(* Logix 5000 project; controller cal1632 1756-L62 rev 16.20; software revision 16.05; part 12 of 57 *)
(* tags used below, declared in another part *)
   AFI : BOOL;
   FAULT : BOOL;
   p01_param_open_oven_temp : REAL;
   p01_param_oven_timer_presets : DINT[32];
   p01_param_process_air_hl : REAL;
   p01_recipe_active : recipe;
   p01_sys_enc : SYS_ENC;
   p01_sys_lc : Limit_Clamp;
   p01r09_open_oven : BOOL;
   p01r09_pb_global_reset : BOOL;
   p01r13_permissive_oxidizer : BOOL;
   p02_dint_from_hmi : hmi_dint;
   p02_real_from_hmi : hmi_real;
   p11_ai_lfl : REAL;
   p11_ai_tc01 : REAL;
   p11_ai_tc02 : REAL;
   p11_ao_cv : REAL;
   p11_di_burner_auto : BOOL;
   p11_di_burner_safeties_ok : BOOL;
   p11_di_exh_flow_ok : BOOL;
   p11_di_flame_failure : BOOL;
   p11_di_flame_on : BOOL;
   p11_di_high_limit_temp_ok : BOOL;
   p11_di_recirc_flow_ok : BOOL;
   p11_di_sp1 : BOOL;
   p11_di_tc01_bo : BOOL;
   p11_di_tc02_bo : BOOL;
   p11_do_enable_burner : BOOL;
   p11_do_rst_flame : BOOL;
   p11_param_fast_to_soak : REAL;
   p11_param_lfl_hhl : REAL;
   p11_param_lfl_hl : REAL;
   p11_param_pid1_ff : REAL;
   p11_param_pid1_kd : REAL;
   p11_param_pid1_ki : REAL;
   p11_param_pid1_kp : REAL;
   p11_param_pid2_ff : REAL;
   p11_param_pid2_kd : REAL;
   p11_param_pid2_ki : REAL;
   p11_param_pid2_kp : REAL;
   p11_param_shutdown_temp : REAL;
   p11_param_soak_to_fast : REAL;
   p11_param_tc01_dev : REAL;
   p11_param_tc01_hl : REAL;
   p11_param_tc01z : REAL;
   p11_param_tc02z : REAL;
   p11_param_zone_pressure : REAL;
   p11r02_shutdown_temp : BOOL;
   p11r02_timer_safe_temp : TIMER[2];
   p11r02_timer_warning : TIMER[4];
   p11r10 : routine;
   p11r10_timer_fault : TIMER[4];
   p11r10_timer_warning : TIMER[4];
   p11r12_Oven_auto_run_on : BOOL;
   p11r16_pid_temp_cv : DINT;
   p11r16_temp_ok : BOOL;
   p11r20 : routine;
   p11r20_safeties_ok : BOOL;
   p11r20_state : DINT;
   p11r20_status : DINT;
   p11r20_timer_fault : TIMER[4];
   p11r20_timer_state_11 : TIMER;
   p11r20_timer_state_3 : TIMER;
   p11r20_timer_state_4 : TIMER;
   p11r20_timer_state_7 : TIMER;
   p11r20_timer_warning : TIMER[4];
   p11r30 : routine;
   p11r30_cv_man_sp : REAL;
   p11r30_pb_auto : BOOL;
   p11r30_pb_manual : BOOL;
   p11r30_pb_zone_off : BOOL;
   p11r30_pb_zone_on : BOOL;
   p11r30_permissive_run : BOOL;
   p11r30_pid_temp : PID;
   p11r30_pid_temp_pv : REAL;
   p11r30_pid_temp_sp : REAL;
   p11r30_pid_temp_sp_error : REAL;
   p11r30_pid_temp_sp_last : REAL;
   p11r30_request_deviation_warning : BOOL;
   p11r30_request_heat : BOOL;
   p11r30_request_heat_last : BOOL;
   p11r30_request_manual : BOOL;
   p11r30_request_PID_shot : BOOL;
   p11r30_request_soak_control : BOOL;
   p11r30_temp_deviation_setpoint : DINT;
   p11r30_timer_fault : TIMER[16];
   p11r30_timer_warning : TIMER[12];
   p11r30_vfds_ok : BOOL;
   p11r31 : routine;
   p11r31_timer_fault : TIMER[5];
   p11r31_timer_warning : TIMER[5];
   p11r32 : routine;
   p11r32_timer_fault : TIMER[5];
   p11r32_timer_warning : TIMER[5];
   p12r30 : routine;
   p23_di_impreg_exhaust_running : BOOL;
   p23_di_impreg_tank_up : BOOL;
   p23r02 : routine;
   p23r13 : routine;
(* P11_Zone_1, continued *)

ROUTINE R10_Parameters   (* ladder *)
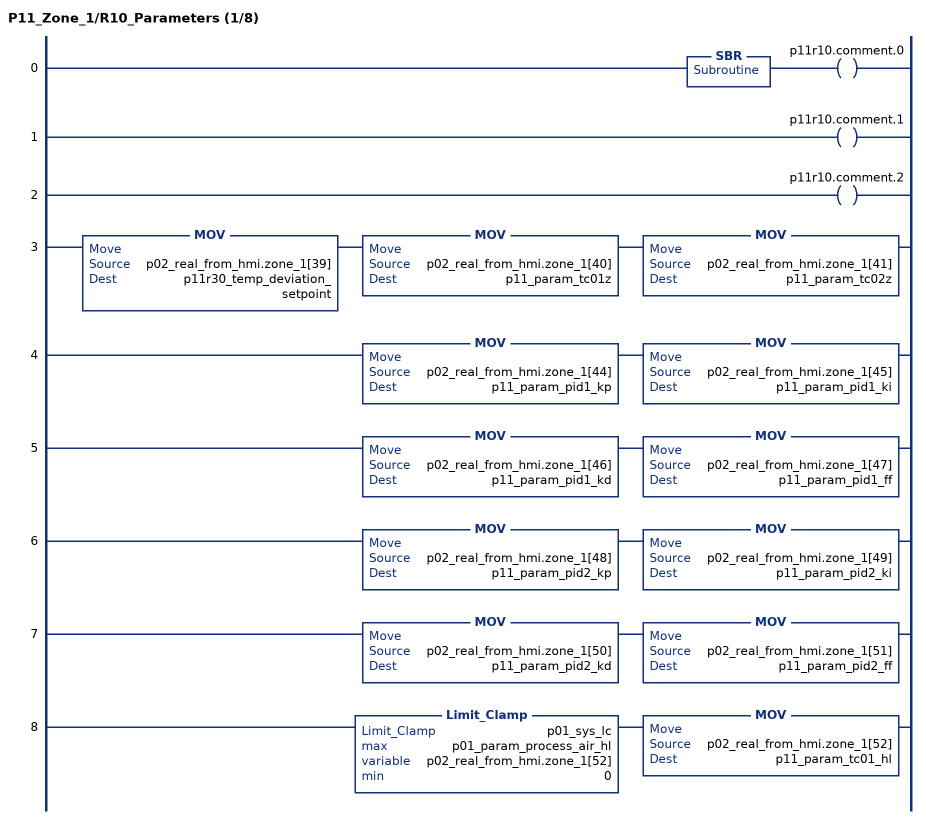
   0: SBR()OTE(p11r10.comment.0);
   1: OTE(p11r10.comment.1);
   2: OTE(p11r10.comment.2);
   3: MOV(p02_real_from_hmi.zone_1[39],p11r30_temp_deviation_setpoint)MOV(p02_real_from_hmi.zone_1[40],p11_param_tc01z)MOV(p02_real_from_hmi.zone_1[41],p11_param_tc02z);
   4: MOV(p02_real_from_hmi.zone_1[44],p11_param_pid1_kp)MOV(p02_real_from_hmi.zone_1[45],p11_param_pid1_ki);
   5: MOV(p02_real_from_hmi.zone_1[46],p11_param_pid1_kd)MOV(p02_real_from_hmi.zone_1[47],p11_param_pid1_ff);
   6: MOV(p02_real_from_hmi.zone_1[48],p11_param_pid2_kp)MOV(p02_real_from_hmi.zone_1[49],p11_param_pid2_ki);
   7: MOV(p02_real_from_hmi.zone_1[50],p11_param_pid2_kd)MOV(p02_real_from_hmi.zone_1[51],p11_param_pid2_ff);
   8: Limit_Clamp(p01_sys_lc,p01_param_process_air_hl,p02_real_from_hmi.zone_1[52],0)MOV(p02_real_from_hmi.zone_1[52],p11_param_tc01_hl);
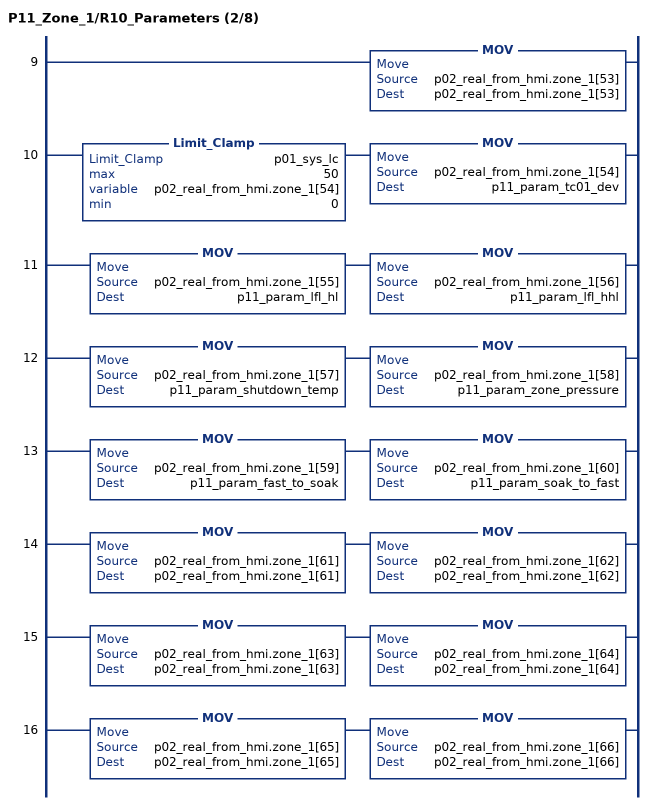
   9: MOV(p02_real_from_hmi.zone_1[53],p02_real_from_hmi.zone_1[53]);
   10: Limit_Clamp(p01_sys_lc,50,p02_real_from_hmi.zone_1[54],0)MOV(p02_real_from_hmi.zone_1[54],p11_param_tc01_dev);
   11: MOV(p02_real_from_hmi.zone_1[55],p11_param_lfl_hl)MOV(p02_real_from_hmi.zone_1[56],p11_param_lfl_hhl);
   12: MOV(p02_real_from_hmi.zone_1[57],p11_param_shutdown_temp)MOV(p02_real_from_hmi.zone_1[58],p11_param_zone_pressure);
   13: MOV(p02_real_from_hmi.zone_1[59],p11_param_fast_to_soak)MOV(p02_real_from_hmi.zone_1[60],p11_param_soak_to_fast);
   14: MOV(p02_real_from_hmi.zone_1[61],p02_real_from_hmi.zone_1[61])MOV(p02_real_from_hmi.zone_1[62],p02_real_from_hmi.zone_1[62]);
   15: MOV(p02_real_from_hmi.zone_1[63],p02_real_from_hmi.zone_1[63])MOV(p02_real_from_hmi.zone_1[64],p02_real_from_hmi.zone_1[64]);
   16: MOV(p02_real_from_hmi.zone_1[65],p02_real_from_hmi.zone_1[65])MOV(p02_real_from_hmi.zone_1[66],p02_real_from_hmi.zone_1[66]);
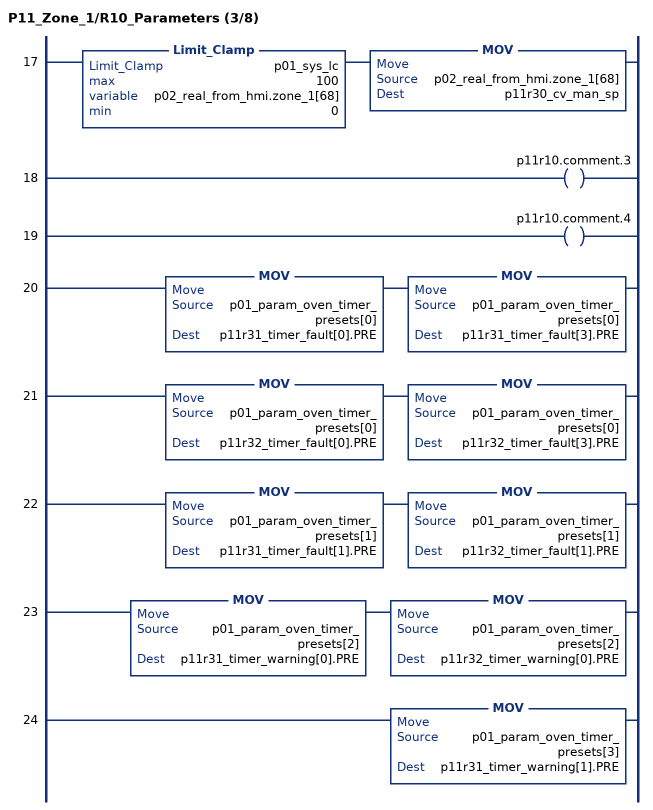
   17: Limit_Clamp(p01_sys_lc,100,p02_real_from_hmi.zone_1[68],0)MOV(p02_real_from_hmi.zone_1[68],p11r30_cv_man_sp);
   18: OTE(p11r10.comment.3);
   19: OTE(p11r10.comment.4);
   20: MOV(p01_param_oven_timer_presets[0],p11r31_timer_fault[0].PRE)MOV(p01_param_oven_timer_presets[0],p11r31_timer_fault[3].PRE);
   21: MOV(p01_param_oven_timer_presets[0],p11r32_timer_fault[0].PRE)MOV(p01_param_oven_timer_presets[0],p11r32_timer_fault[3].PRE);
   22: MOV(p01_param_oven_timer_presets[1],p11r31_timer_fault[1].PRE)MOV(p01_param_oven_timer_presets[1],p11r32_timer_fault[1].PRE);
   23: MOV(p01_param_oven_timer_presets[2],p11r31_timer_warning[0].PRE)MOV(p01_param_oven_timer_presets[2],p11r32_timer_warning[0].PRE);
   24: MOV(p01_param_oven_timer_presets[3],p11r31_timer_warning[1].PRE);
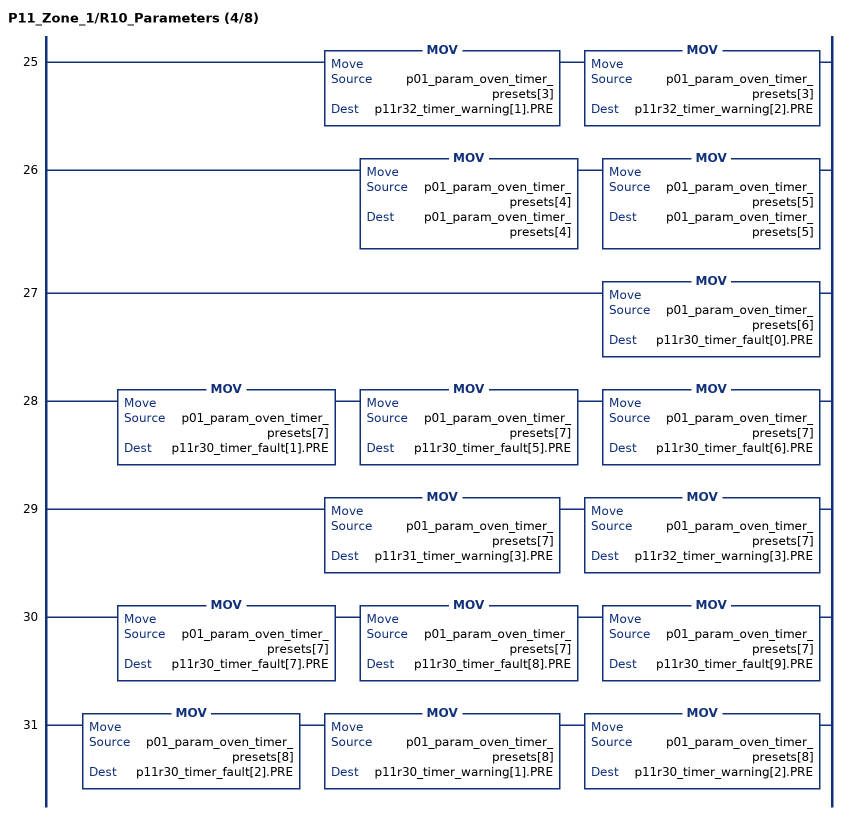
   25: MOV(p01_param_oven_timer_presets[3],p11r32_timer_warning[1].PRE)MOV(p01_param_oven_timer_presets[3],p11r32_timer_warning[2].PRE);
   26: MOV(p01_param_oven_timer_presets[4],p01_param_oven_timer_presets[4])MOV(p01_param_oven_timer_presets[5],p01_param_oven_timer_presets[5]);
   27: MOV(p01_param_oven_timer_presets[6],p11r30_timer_fault[0].PRE);
   28: MOV(p01_param_oven_timer_presets[7],p11r30_timer_fault[1].PRE)MOV(p01_param_oven_timer_presets[7],p11r30_timer_fault[5].PRE)MOV(p01_param_oven_timer_presets[7],p11r30_timer_fault[6].PRE);
   29: MOV(p01_param_oven_timer_presets[7],p11r31_timer_warning[3].PRE)MOV(p01_param_oven_timer_presets[7],p11r32_timer_warning[3].PRE);
   30: MOV(p01_param_oven_timer_presets[7],p11r30_timer_fault[7].PRE)MOV(p01_param_oven_timer_presets[7],p11r30_timer_fault[8].PRE)MOV(p01_param_oven_timer_presets[7],p11r30_timer_fault[9].PRE);
   31: MOV(p01_param_oven_timer_presets[8],p11r30_timer_fault[2].PRE)MOV(p01_param_oven_timer_presets[8],p11r30_timer_warning[1].PRE)MOV(p01_param_oven_timer_presets[8],p11r30_timer_warning[2].PRE);
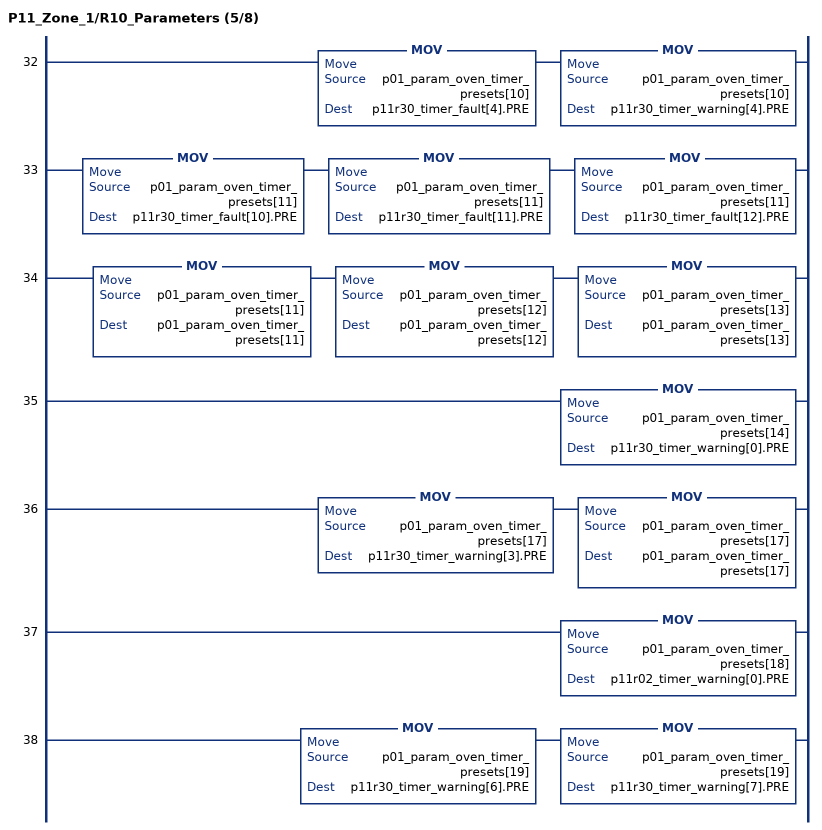
   32: MOV(p01_param_oven_timer_presets[10],p11r30_timer_fault[4].PRE)MOV(p01_param_oven_timer_presets[10],p11r30_timer_warning[4].PRE);
   33: MOV(p01_param_oven_timer_presets[11],p11r30_timer_fault[10].PRE)MOV(p01_param_oven_timer_presets[11],p11r30_timer_fault[11].PRE)MOV(p01_param_oven_timer_presets[11],p11r30_timer_fault[12].PRE);
   34: MOV(p01_param_oven_timer_presets[11],p01_param_oven_timer_presets[11])MOV(p01_param_oven_timer_presets[12],p01_param_oven_timer_presets[12])MOV(p01_param_oven_timer_presets[13],p01_param_oven_timer_presets[13]);
   35: MOV(p01_param_oven_timer_presets[14],p11r30_timer_warning[0].PRE);
   36: MOV(p01_param_oven_timer_presets[17],p11r30_timer_warning[3].PRE)MOV(p01_param_oven_timer_presets[17],p01_param_oven_timer_presets[17]);
   37: MOV(p01_param_oven_timer_presets[18],p11r02_timer_warning[0].PRE);
   38: MOV(p01_param_oven_timer_presets[19],p11r30_timer_warning[6].PRE)MOV(p01_param_oven_timer_presets[19],p11r30_timer_warning[7].PRE);
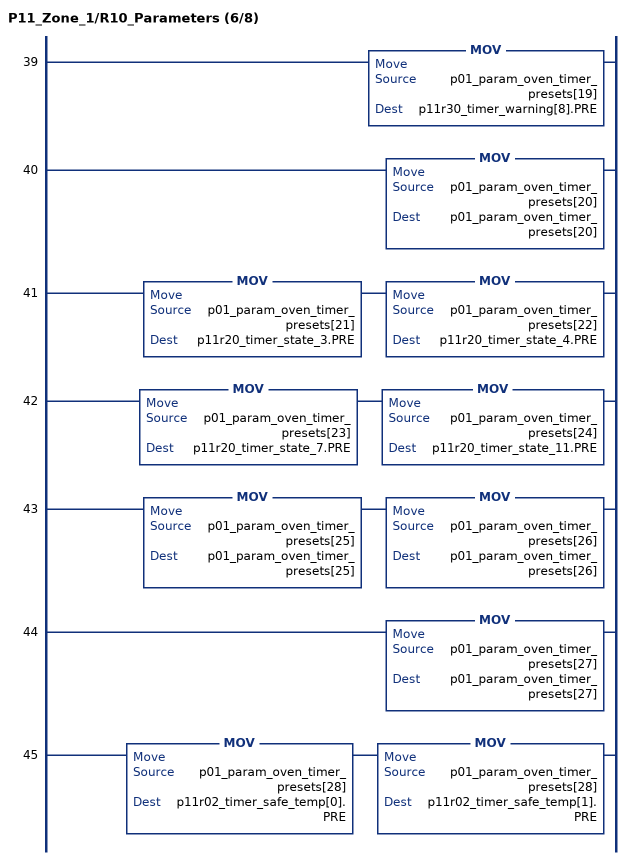
   39: MOV(p01_param_oven_timer_presets[19],p11r30_timer_warning[8].PRE);
   40: MOV(p01_param_oven_timer_presets[20],p01_param_oven_timer_presets[20]);
   41: MOV(p01_param_oven_timer_presets[21],p11r20_timer_state_3.PRE)MOV(p01_param_oven_timer_presets[22],p11r20_timer_state_4.PRE);
   42: MOV(p01_param_oven_timer_presets[23],p11r20_timer_state_7.PRE)MOV(p01_param_oven_timer_presets[24],p11r20_timer_state_11.PRE);
   43: MOV(p01_param_oven_timer_presets[25],p01_param_oven_timer_presets[25])MOV(p01_param_oven_timer_presets[26],p01_param_oven_timer_presets[26]);
   44: MOV(p01_param_oven_timer_presets[27],p01_param_oven_timer_presets[27]);
   45: MOV(p01_param_oven_timer_presets[28],p11r02_timer_safe_temp[0].PRE)MOV(p01_param_oven_timer_presets[28],p11r02_timer_safe_temp[1].PRE);
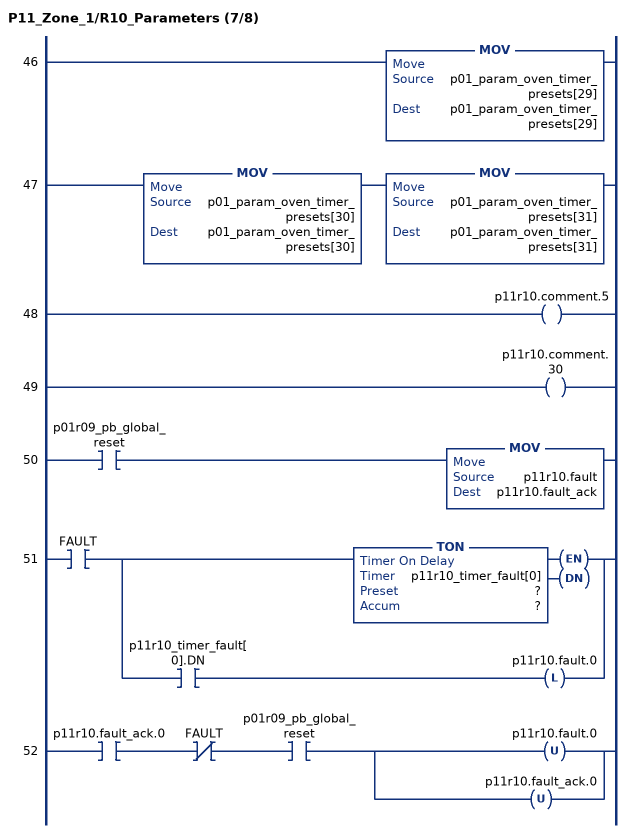
   46: MOV(p01_param_oven_timer_presets[29],p01_param_oven_timer_presets[29]);
   47: MOV(p01_param_oven_timer_presets[30],p01_param_oven_timer_presets[30])MOV(p01_param_oven_timer_presets[31],p01_param_oven_timer_presets[31]);
   48: OTE(p11r10.comment.5);
   49: OTE(p11r10.comment.30);
   50: XIC(p01r09_pb_global_reset)MOV(p11r10.fault,p11r10.fault_ack);
   51: XIC(FAULT)[TON(p11r10_timer_fault[0],?,?) ,XIC(p11r10_timer_fault[0].DN) OTL(p11r10.fault.0) ];
   52: XIC(p11r10.fault_ack.0)XIO(FAULT)XIC(p01r09_pb_global_reset)[OTU(p11r10.fault.0) ,OTU(p11r10.fault_ack.0) ];
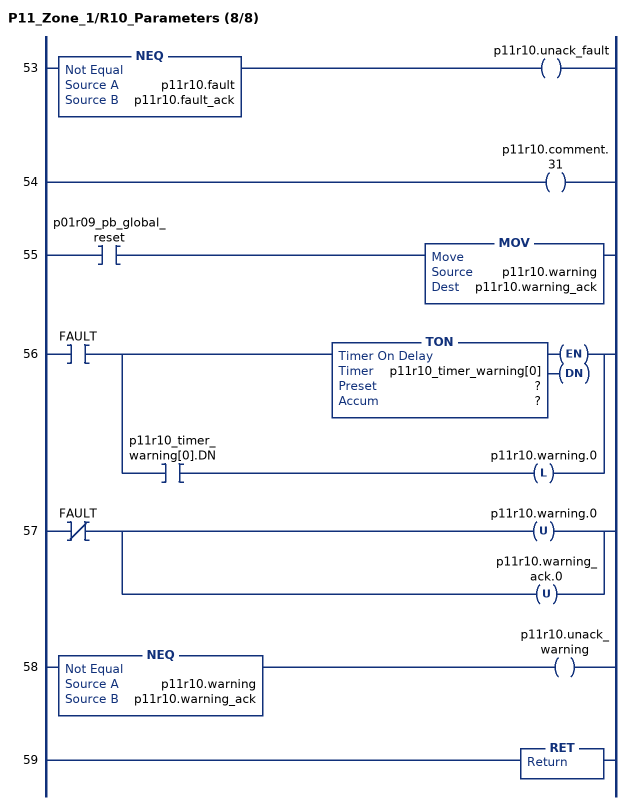
   53: NEQ(p11r10.fault,p11r10.fault_ack)OTE(p11r10.unack_fault);
   54: OTE(p11r10.comment.31);
   55: XIC(p01r09_pb_global_reset)MOV(p11r10.warning,p11r10.warning_ack);
   56: XIC(FAULT)[TON(p11r10_timer_warning[0],?,?) ,XIC(p11r10_timer_warning[0].DN) OTL(p11r10.warning.0) ];
   57: XIO(FAULT)[OTU(p11r10.warning.0) ,OTU(p11r10.warning_ack.0) ];
   58: NEQ(p11r10.warning,p11r10.warning_ack)OTE(p11r10.unack_warning);
   59: RET();
END_ROUTINE

ROUTINE R20_Temp_Sequence   (* ladder *)
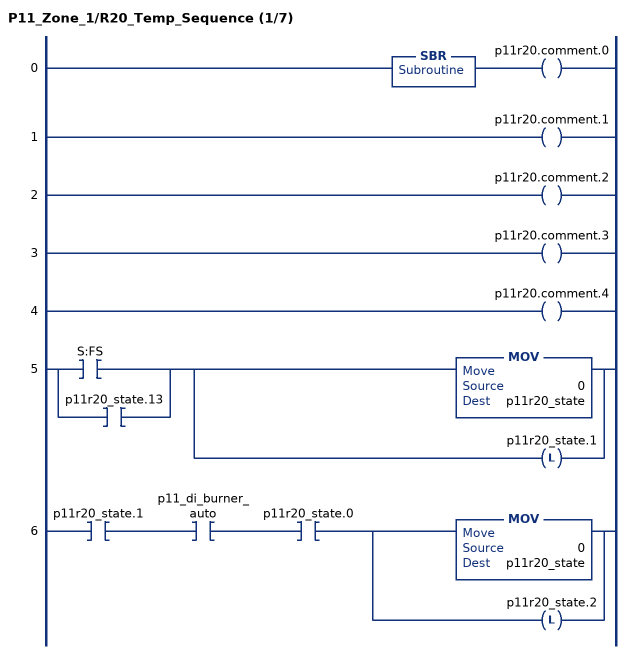
   0: SBR()OTE(p11r20.comment.0);
   1: OTE(p11r20.comment.1);
   2: OTE(p11r20.comment.2);
   3: OTE(p11r20.comment.3);
   4: OTE(p11r20.comment.4);
   5: [XIC(S:FS) ,XIC(p11r20_state.13) ][MOV(0,p11r20_state) ,OTL(p11r20_state.1) ];
   6: XIC(p11r20_state.1)XIC(p11_di_burner_auto)XIC(p11r20_state.0)[MOV(0,p11r20_state) ,OTL(p11r20_state.2) ];
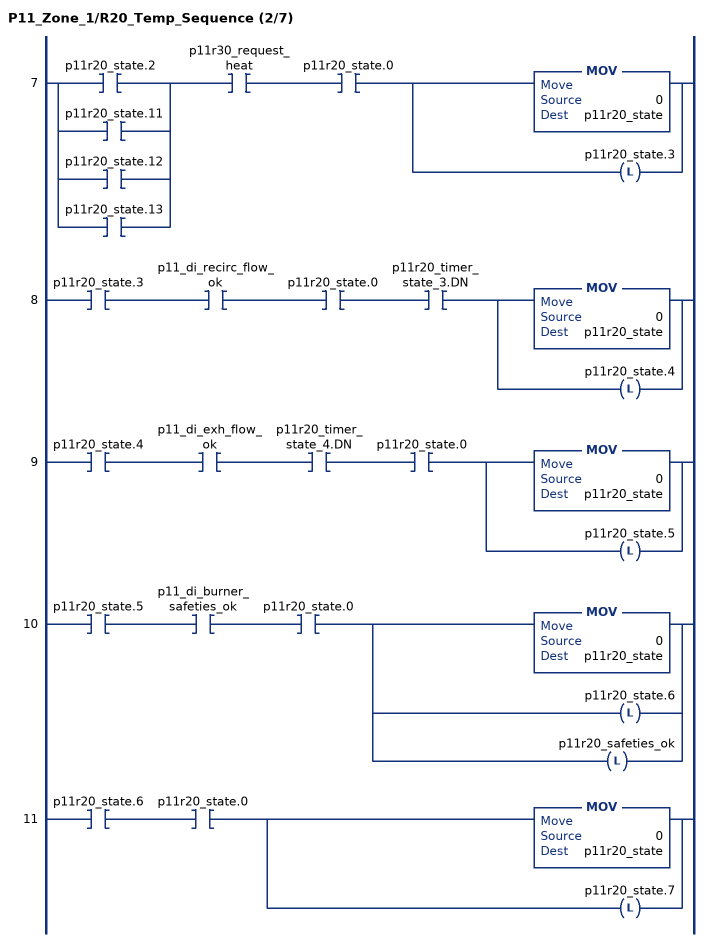
   7: [XIC(p11r20_state.2) ,XIC(p11r20_state.11) ,XIC(p11r20_state.12) ,XIC(p11r20_state.13) ]XIC(p11r30_request_heat)XIC(p11r20_state.0)[MOV(0,p11r20_state) ,OTL(p11r20_state.3) ];
   8: XIC(p11r20_state.3)XIC(p11_di_recirc_flow_ok)XIC(p11r20_state.0)XIC(p11r20_timer_state_3.DN)[MOV(0,p11r20_state) ,OTL(p11r20_state.4) ];
   9: XIC(p11r20_state.4)XIC(p11_di_exh_flow_ok)XIC(p11r20_timer_state_4.DN)XIC(p11r20_state.0)[MOV(0,p11r20_state) ,OTL(p11r20_state.5) ];
   10: XIC(p11r20_state.5)XIC(p11_di_burner_safeties_ok)XIC(p11r20_state.0)[MOV(0,p11r20_state) ,OTL(p11r20_state.6) ,OTL(p11r20_safeties_ok) ];
   11: XIC(p11r20_state.6)XIC(p11r20_state.0)[MOV(0,p11r20_state) ,OTL(p11r20_state.7) ];
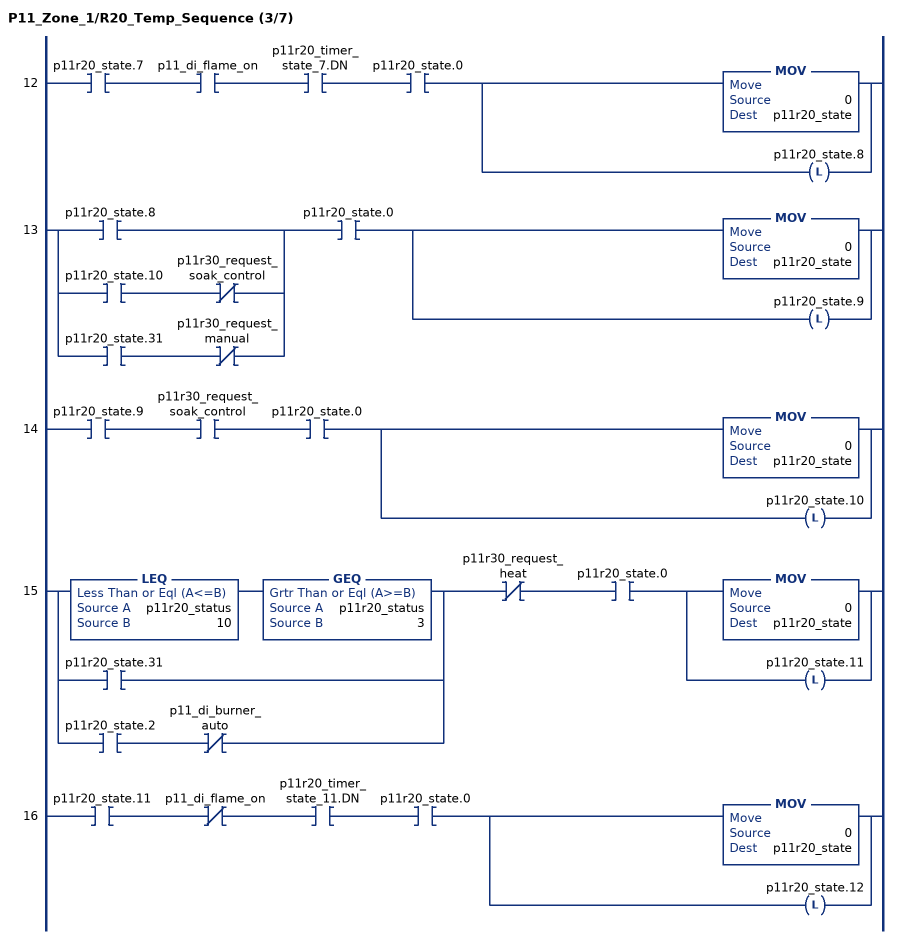
   12: XIC(p11r20_state.7)XIC(p11_di_flame_on)XIC(p11r20_timer_state_7.DN)XIC(p11r20_state.0)[MOV(0,p11r20_state) ,OTL(p11r20_state.8) ];
   13: [XIC(p11r20_state.8) ,XIC(p11r20_state.10) XIO(p11r30_request_soak_control) ,XIC(p11r20_state.31) XIO(p11r30_request_manual) ]XIC(p11r20_state.0)[MOV(0,p11r20_state) ,OTL(p11r20_state.9) ];
   14: XIC(p11r20_state.9)XIC(p11r30_request_soak_control)XIC(p11r20_state.0)[MOV(0,p11r20_state) ,OTL(p11r20_state.10) ];
   15: [[LEQ(p11r20_status,10) GEQ(p11r20_status,3) ,XIC(p11r20_state.31) ] ,XIC(p11r20_state.2) XIO(p11_di_burner_auto) ]XIO(p11r30_request_heat)XIC(p11r20_state.0)[MOV(0,p11r20_state) ,OTL(p11r20_state.11) ];
   16: XIC(p11r20_state.11)XIO(p11_di_flame_on)XIC(p11r20_timer_state_11.DN)XIC(p11r20_state.0)[MOV(0,p11r20_state) ,OTL(p11r20_state.12) ];
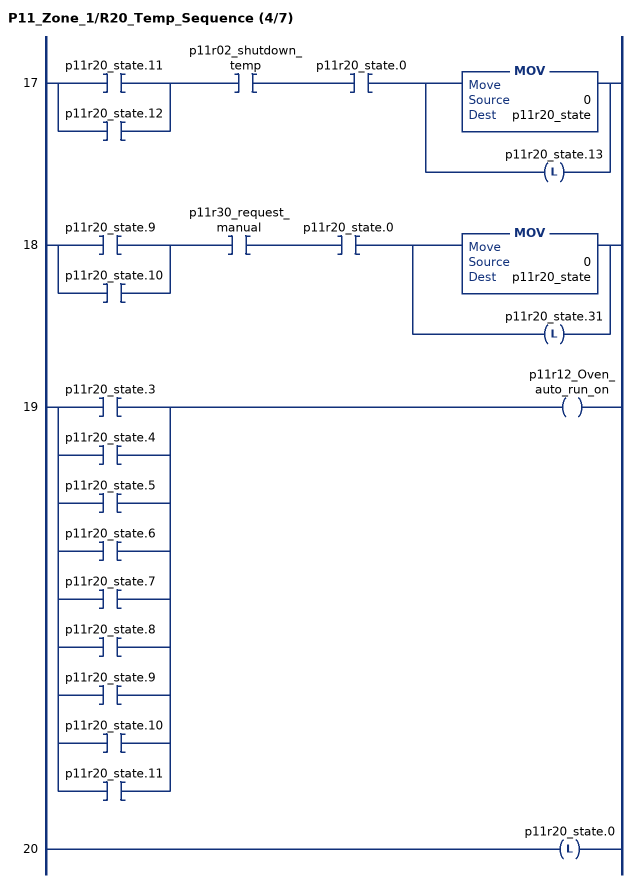
   17: [XIC(p11r20_state.11) ,XIC(p11r20_state.12) ]XIC(p11r02_shutdown_temp)XIC(p11r20_state.0)[MOV(0,p11r20_state) ,OTL(p11r20_state.13) ];
   18: [XIC(p11r20_state.9) ,XIC(p11r20_state.10) ]XIC(p11r30_request_manual)XIC(p11r20_state.0)[MOV(0,p11r20_state) ,OTL(p11r20_state.31) ];
   19: [XIC(p11r20_state.3) ,XIC(p11r20_state.4) ,XIC(p11r20_state.5) ,XIC(p11r20_state.6) ,XIC(p11r20_state.7) ,XIC(p11r20_state.8) ,XIC(p11r20_state.9) ,XIC(p11r20_state.10) ,XIC(p11r20_state.11) ]OTE(p11r12_Oven_auto_run_on);
   20: OTL(p11r20_state.0);
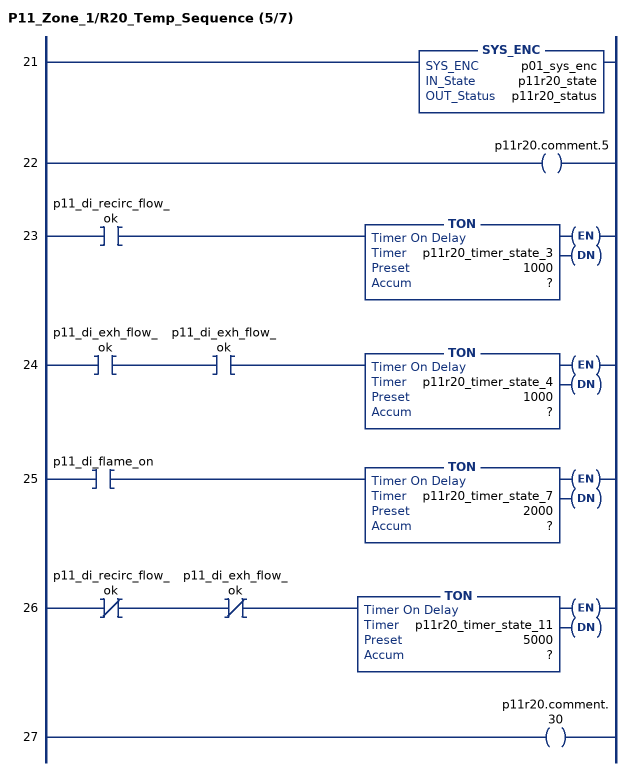
   21: SYS_ENC(p01_sys_enc,p11r20_state,p11r20_status);
   22: OTE(p11r20.comment.5);
   23: XIC(p11_di_recirc_flow_ok)TON(p11r20_timer_state_3,?,?);
   24: XIC(p11_di_exh_flow_ok)XIC(p11_di_exh_flow_ok)TON(p11r20_timer_state_4,?,?);
   25: XIC(p11_di_flame_on)TON(p11r20_timer_state_7,?,?);
   26: XIO(p11_di_recirc_flow_ok)XIO(p11_di_exh_flow_ok)TON(p11r20_timer_state_11,?,?);
   27: OTE(p11r20.comment.30);
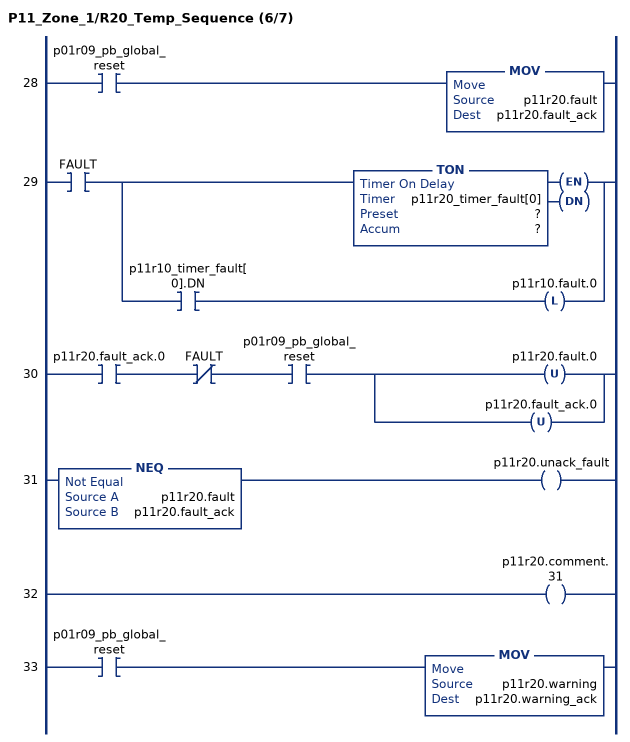
   28: XIC(p01r09_pb_global_reset)MOV(p11r20.fault,p11r20.fault_ack);
   29: XIC(FAULT)[TON(p11r20_timer_fault[0],?,?) ,XIC(p11r10_timer_fault[0].DN) OTL(p11r10.fault.0) ];
   30: XIC(p11r20.fault_ack.0)XIO(FAULT)XIC(p01r09_pb_global_reset)[OTU(p11r20.fault.0) ,OTU(p11r20.fault_ack.0) ];
   31: NEQ(p11r20.fault,p11r20.fault_ack)OTE(p11r20.unack_fault);
   32: OTE(p11r20.comment.31);
   33: XIC(p01r09_pb_global_reset)MOV(p11r20.warning,p11r20.warning_ack);
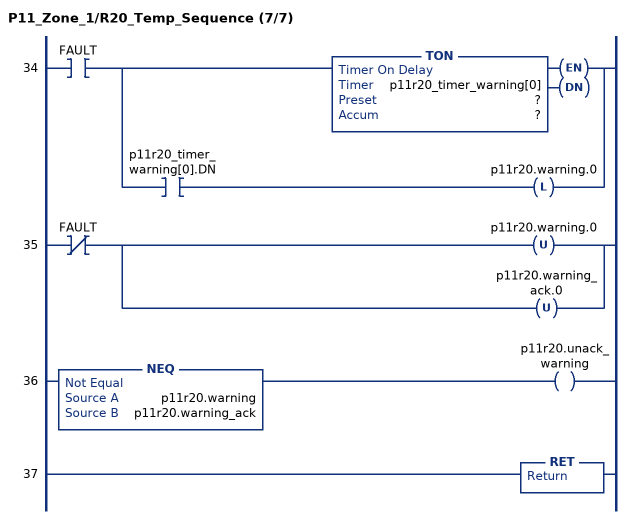
   34: XIC(FAULT)[TON(p11r20_timer_warning[0],?,?) ,XIC(p11r20_timer_warning[0].DN) OTL(p11r20.warning.0) ];
   35: XIO(FAULT)[OTU(p11r20.warning.0) ,OTU(p11r20.warning_ack.0) ];
   36: NEQ(p11r20.warning,p11r20.warning_ack)OTE(p11r20.unack_warning);
   37: RET();
END_ROUTINE

ROUTINE R30_Temperature_Control   (* ladder *)
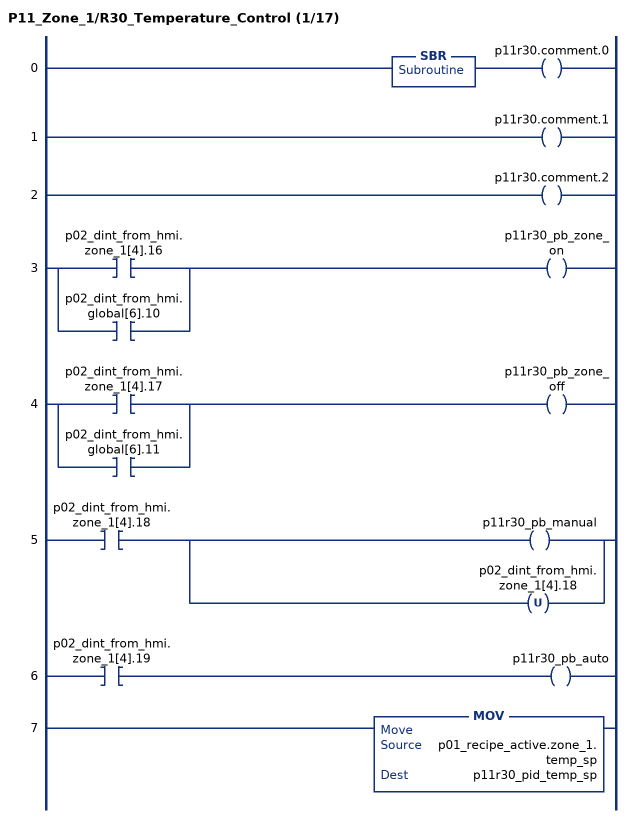
   0: SBR()OTE(p11r30.comment.0);
   1: OTE(p11r30.comment.1);
   2: OTE(p11r30.comment.2);
   3: [XIC(p02_dint_from_hmi.zone_1[4].16) ,XIC(p02_dint_from_hmi.global[6].10) ]OTE(p11r30_pb_zone_on);
   4: [XIC(p02_dint_from_hmi.zone_1[4].17) ,XIC(p02_dint_from_hmi.global[6].11) ]OTE(p11r30_pb_zone_off);
   5: XIC(p02_dint_from_hmi.zone_1[4].18)[OTE(p11r30_pb_manual) ,OTU(p02_dint_from_hmi.zone_1[4].18) ];
   6: XIC(p02_dint_from_hmi.zone_1[4].19)OTE(p11r30_pb_auto);
   7: MOV(p01_recipe_active.zone_1.temp_sp,p11r30_pid_temp_sp);
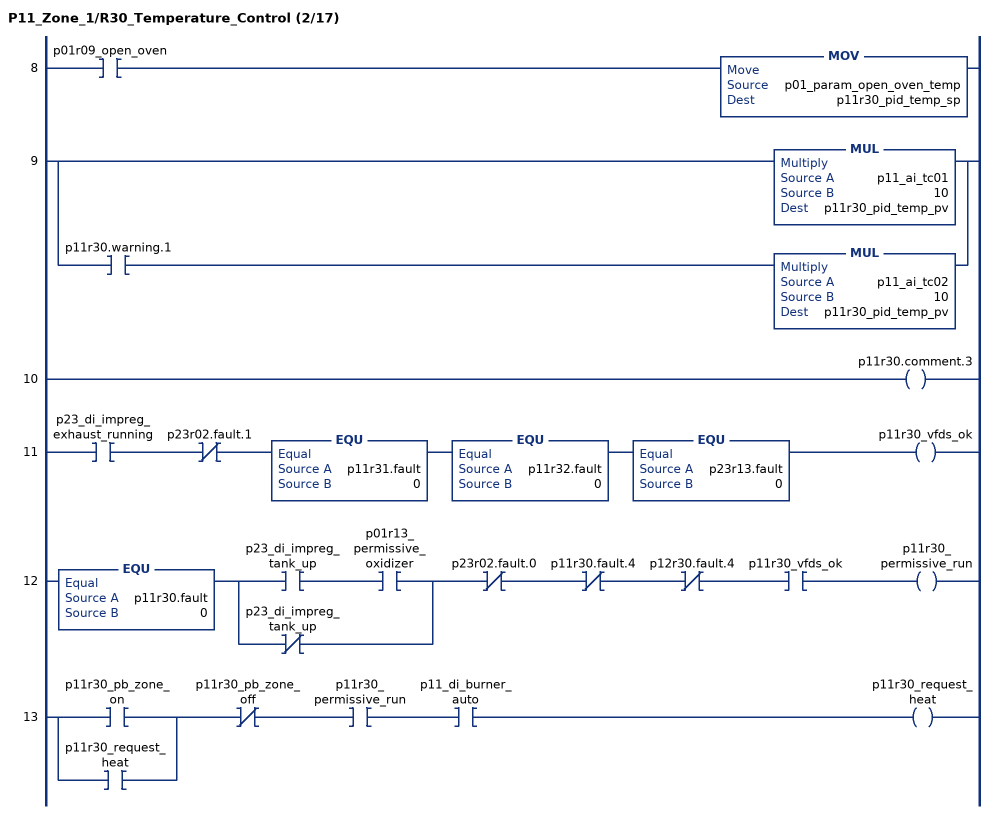
   8: XIC(p01r09_open_oven)MOV(p01_param_open_oven_temp,p11r30_pid_temp_sp);
   9: [MUL(p11_ai_tc01,10,p11r30_pid_temp_pv) ,XIC(p11r30.warning.1) MUL(p11_ai_tc02,10,p11r30_pid_temp_pv) ];
   10: OTE(p11r30.comment.3);
   11: XIC(p23_di_impreg_exhaust_running)XIO(p23r02.fault.1)EQU(p11r31.fault,0)EQU(p11r32.fault,0)EQU(p23r13.fault,0)OTE(p11r30_vfds_ok);
   12: EQU(p11r30.fault,0)[XIC(p23_di_impreg_tank_up) XIC(p01r13_permissive_oxidizer) ,XIO(p23_di_impreg_tank_up) ]XIO(p23r02.fault.0)XIO(p11r30.fault.4)XIO(p12r30.fault.4)XIC(p11r30_vfds_ok)OTE(p11r30_permissive_run);
   13: [XIC(p11r30_pb_zone_on) ,XIC(p11r30_request_heat) ]XIO(p11r30_pb_zone_off)XIC(p11r30_permissive_run)XIC(p11_di_burner_auto)OTE(p11r30_request_heat);
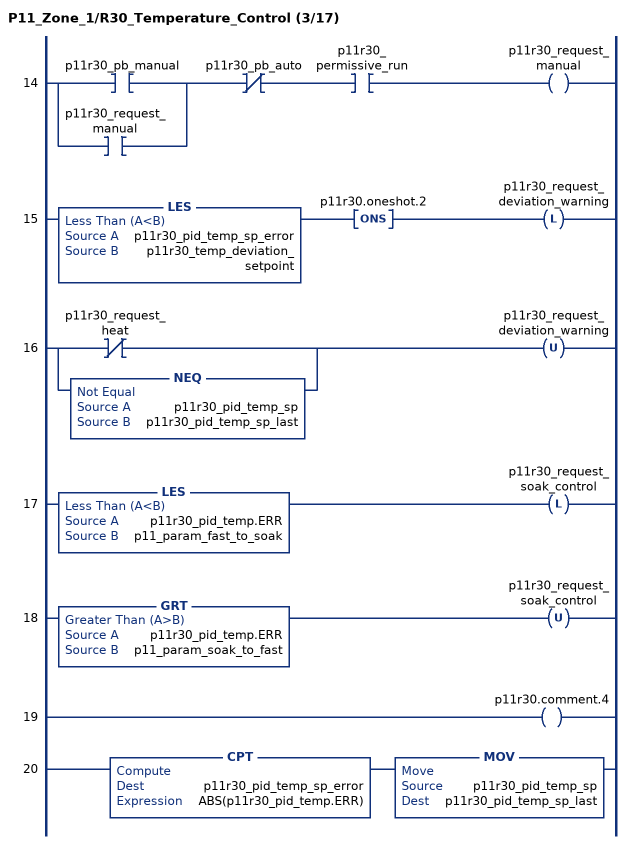
   14: [XIC(p11r30_pb_manual) ,XIC(p11r30_request_manual) ]XIO(p11r30_pb_auto)XIC(p11r30_permissive_run)OTE(p11r30_request_manual);
   15: LES(p11r30_pid_temp_sp_error,p11r30_temp_deviation_setpoint)ONS(p11r30.oneshot.2)OTL(p11r30_request_deviation_warning);
   16: [XIO(p11r30_request_heat) ,NEQ(p11r30_pid_temp_sp,p11r30_pid_temp_sp_last) ]OTU(p11r30_request_deviation_warning);
   17: LES(p11r30_pid_temp.ERR,p11_param_fast_to_soak)OTL(p11r30_request_soak_control);
   18: GRT(p11r30_pid_temp.ERR,p11_param_soak_to_fast)OTU(p11r30_request_soak_control);
   19: OTE(p11r30.comment.4);
   20: CPT(p11r30_pid_temp_sp_error,ABS(p11r30_pid_temp.ERR))MOV(p11r30_pid_temp_sp,p11r30_pid_temp_sp_last);
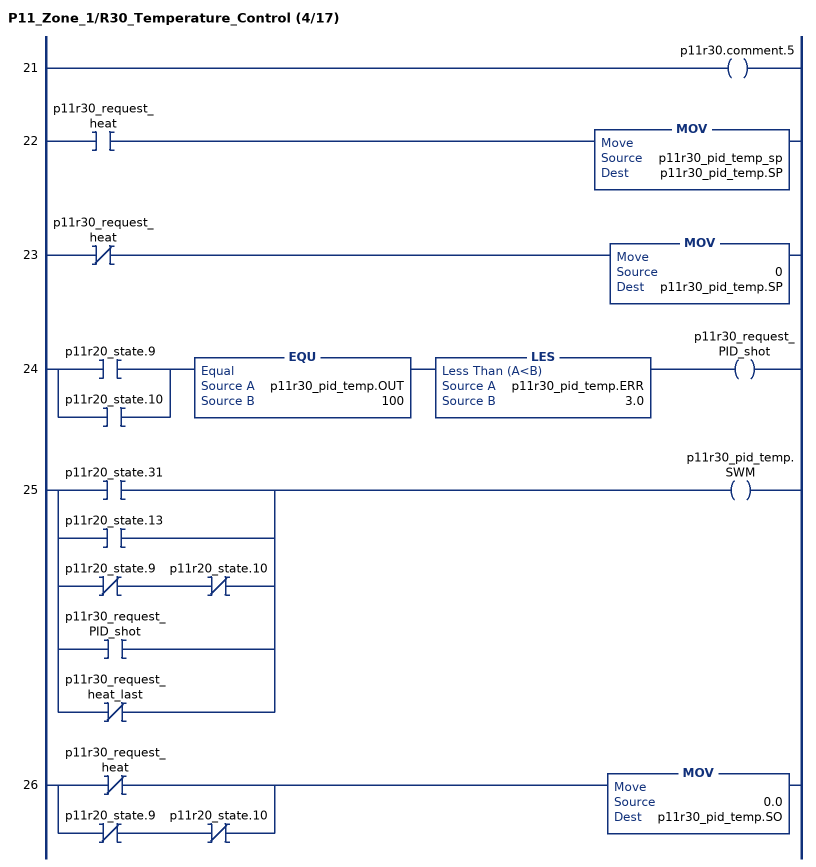
   21: OTE(p11r30.comment.5);
   22: XIC(p11r30_request_heat)MOV(p11r30_pid_temp_sp,p11r30_pid_temp.SP);
   23: XIO(p11r30_request_heat)MOV(0,p11r30_pid_temp.SP);
   24: [XIC(p11r20_state.9) ,XIC(p11r20_state.10) ]EQU(p11r30_pid_temp.OUT,100)LES(p11r30_pid_temp.ERR,3.0)OTE(p11r30_request_PID_shot);
   25: [XIC(p11r20_state.31) ,XIC(p11r20_state.13) ,XIO(p11r20_state.9) XIO(p11r20_state.10) ,XIC(p11r30_request_PID_shot) ,XIO(p11r30_request_heat_last) ]OTE(p11r30_pid_temp.SWM);
   26: [XIO(p11r30_request_heat) ,XIO(p11r20_state.9) XIO(p11r20_state.10) ]MOV(0.0,p11r30_pid_temp.SO);
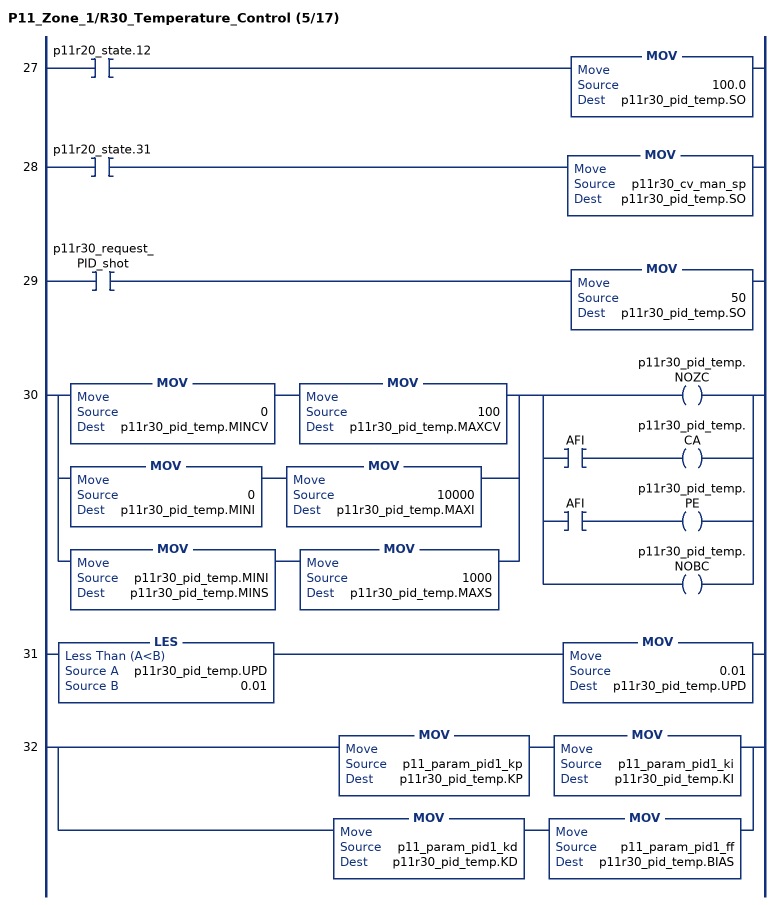
   27: XIC(p11r20_state.12)MOV(100.0,p11r30_pid_temp.SO);
   28: XIC(p11r20_state.31)MOV(p11r30_cv_man_sp,p11r30_pid_temp.SO);
   29: XIC(p11r30_request_PID_shot)MOV(50,p11r30_pid_temp.SO);
   30: [MOV(0,p11r30_pid_temp.MINCV) MOV(100,p11r30_pid_temp.MAXCV) ,MOV(0,p11r30_pid_temp.MINI) MOV(10000,p11r30_pid_temp.MAXI) ,MOV(p11r30_pid_temp.MINI,p11r30_pid_temp.MINS) MOV(1000,p11r30_pid_temp.MAXS) ][OTE(p11r30_pid_temp.NOZC) ,XIC(AFI) OTE(p11r30_pid_temp.CA) ,XIC(AFI) OTE(p11r30_pid_temp.PE) ,OTE(p11r30_pid_temp.NOBC) ];
   31: LES(p11r30_pid_temp.UPD,0.01)MOV(0.01,p11r30_pid_temp.UPD);
   32: [MOV(p11_param_pid1_kp,p11r30_pid_temp.KP) MOV(p11_param_pid1_ki,p11r30_pid_temp.KI) ,MOV(p11_param_pid1_kd,p11r30_pid_temp.KD) MOV(p11_param_pid1_ff,p11r30_pid_temp.BIAS) ];
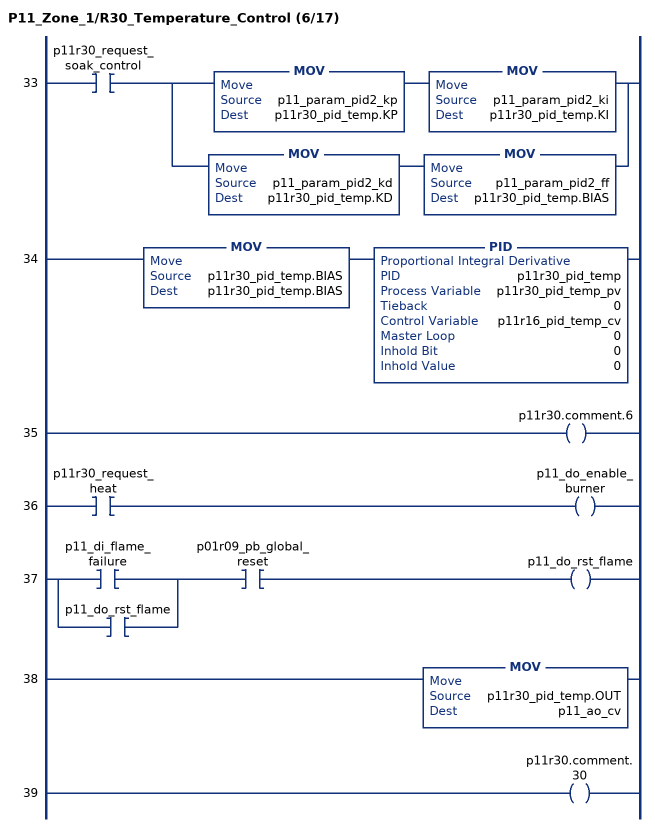
   33: XIC(p11r30_request_soak_control)[MOV(p11_param_pid2_kp,p11r30_pid_temp.KP) MOV(p11_param_pid2_ki,p11r30_pid_temp.KI) ,MOV(p11_param_pid2_kd,p11r30_pid_temp.KD) MOV(p11_param_pid2_ff,p11r30_pid_temp.BIAS) ];
   34: MOV(p11r30_pid_temp.BIAS,p11r30_pid_temp.BIAS)PID(p11r30_pid_temp,p11r30_pid_temp_pv,0,p11r16_pid_temp_cv,0,0,0);
   35: OTE(p11r30.comment.6);
   36: XIC(p11r30_request_heat)OTE(p11_do_enable_burner);
   37: [XIC(p11_di_flame_failure) ,XIC(p11_do_rst_flame) ]XIC(p01r09_pb_global_reset)OTE(p11_do_rst_flame);
   38: MOV(p11r30_pid_temp.OUT,p11_ao_cv);
   39: OTE(p11r30.comment.30);
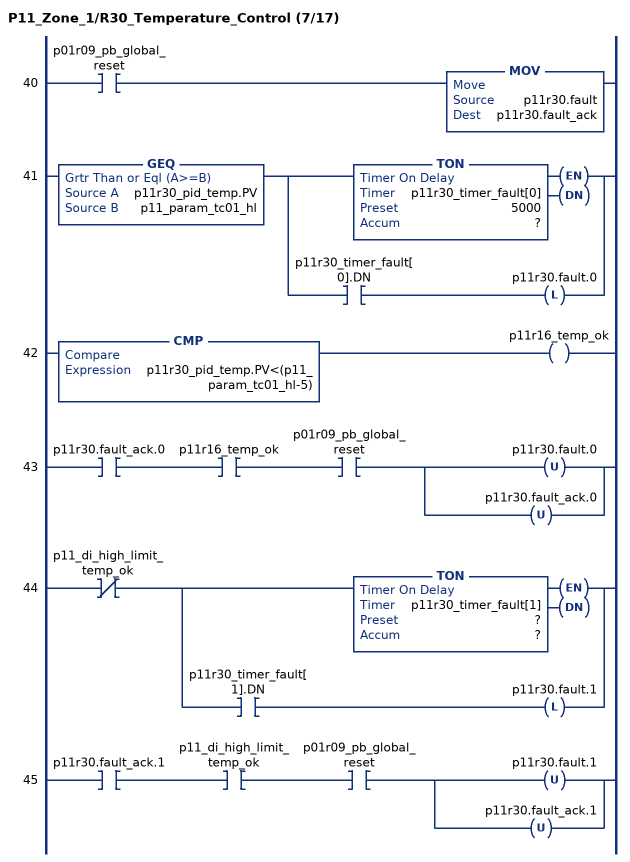
   40: XIC(p01r09_pb_global_reset)MOV(p11r30.fault,p11r30.fault_ack);
   41: GEQ(p11r30_pid_temp.PV,p11_param_tc01_hl)[TON(p11r30_timer_fault[0],?,?) ,XIC(p11r30_timer_fault[0].DN) OTL(p11r30.fault.0) ];
   42: CMP(p11r30_pid_temp.PV<(p11_param_tc01_hl-5))OTE(p11r16_temp_ok);
   43: XIC(p11r30.fault_ack.0)XIC(p11r16_temp_ok)XIC(p01r09_pb_global_reset)[OTU(p11r30.fault.0) ,OTU(p11r30.fault_ack.0) ];
   44: XIO(p11_di_high_limit_temp_ok)[TON(p11r30_timer_fault[1],?,?) ,XIC(p11r30_timer_fault[1].DN) OTL(p11r30.fault.1) ];
   45: XIC(p11r30.fault_ack.1)XIC(p11_di_high_limit_temp_ok)XIC(p01r09_pb_global_reset)[OTU(p11r30.fault.1) ,OTU(p11r30.fault_ack.1) ];
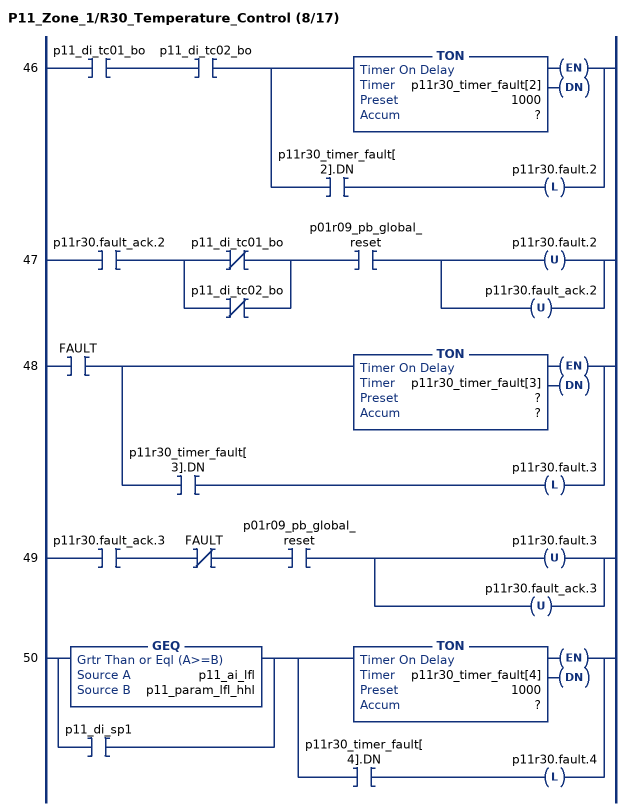
   46: XIC(p11_di_tc01_bo)XIC(p11_di_tc02_bo)[TON(p11r30_timer_fault[2],?,?) ,XIC(p11r30_timer_fault[2].DN) OTL(p11r30.fault.2) ];
   47: XIC(p11r30.fault_ack.2)[XIO(p11_di_tc01_bo) ,XIO(p11_di_tc02_bo) ]XIC(p01r09_pb_global_reset)[OTU(p11r30.fault.2) ,OTU(p11r30.fault_ack.2) ];
   48: XIC(FAULT)[TON(p11r30_timer_fault[3],?,?) ,XIC(p11r30_timer_fault[3].DN) OTL(p11r30.fault.3) ];
   49: XIC(p11r30.fault_ack.3)XIO(FAULT)XIC(p01r09_pb_global_reset)[OTU(p11r30.fault.3) ,OTU(p11r30.fault_ack.3) ];
   50: [GEQ(p11_ai_lfl,p11_param_lfl_hhl) ,XIC(p11_di_sp1) ][TON(p11r30_timer_fault[4],?,?) ,XIC(p11r30_timer_fault[4].DN) OTL(p11r30.fault.4) ];
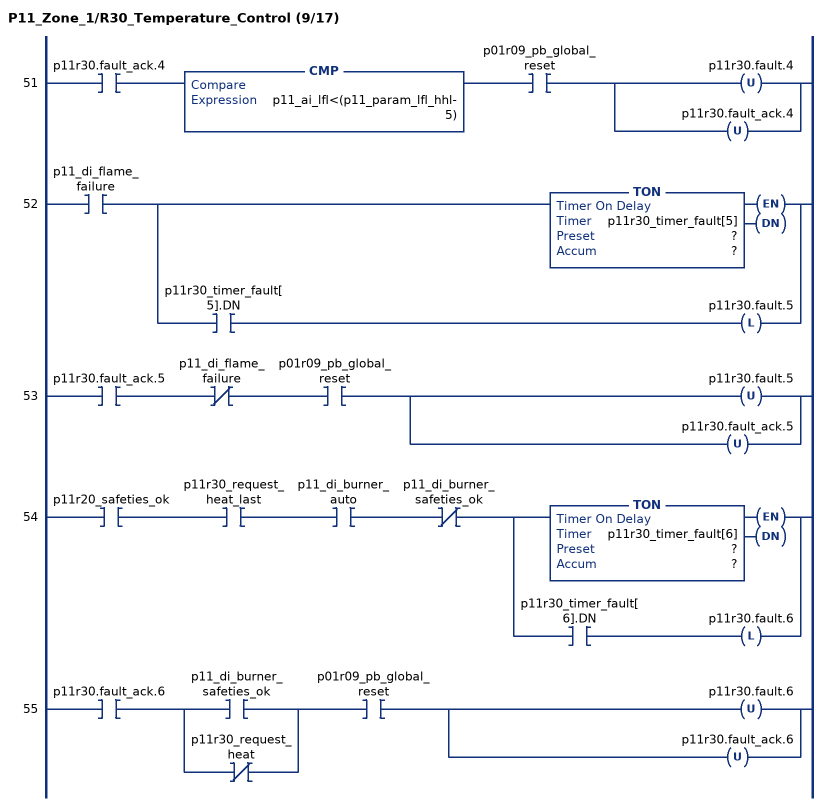
   51: XIC(p11r30.fault_ack.4)CMP(p11_ai_lfl<(p11_param_lfl_hhl-5))XIC(p01r09_pb_global_reset)[OTU(p11r30.fault.4) ,OTU(p11r30.fault_ack.4) ];
   52: XIC(p11_di_flame_failure)[TON(p11r30_timer_fault[5],?,?) ,XIC(p11r30_timer_fault[5].DN) OTL(p11r30.fault.5) ];
   53: XIC(p11r30.fault_ack.5)XIO(p11_di_flame_failure)XIC(p01r09_pb_global_reset)[OTU(p11r30.fault.5) ,OTU(p11r30.fault_ack.5) ];
   54: XIC(p11r20_safeties_ok)XIC(p11r30_request_heat_last)XIC(p11_di_burner_auto)XIO(p11_di_burner_safeties_ok)[TON(p11r30_timer_fault[6],?,?) ,XIC(p11r30_timer_fault[6].DN) OTL(p11r30.fault.6) ];
   55: XIC(p11r30.fault_ack.6)[XIC(p11_di_burner_safeties_ok) ,XIO(p11r30_request_heat) ]XIC(p01r09_pb_global_reset)[OTU(p11r30.fault.6) ,OTU(p11r30.fault_ack.6) ];
